Fanuc KAREL source: FanucServiceLib.kl

PROGRAM FANUC_SERVICE_LIB
%NOLOCKGROUP
%NOPAUSE = ERROR + COMMAND + TPENABLE
%NOABORT = ERROR + COMMAND
%COMMENT = 'Shared helpers for resident service'
%ENVIRONMENT sysdef
%ENVIRONMENT kclop
%ENVIRONMENT fdev
%ENVIRONMENT MOTN
%ENVIRONMENT REGOPE
%ENVIRONMENT MULTI
%ENVIRONMENT STRNG

VAR
  g_status  : INTEGER
  g_entry   : INTEGER
  g_bool    : BOOLEAN
  g_int     : INTEGER
  g_real    : REAL
  g_state_real : REAL
  g_state_is_real : BOOLEAN
  g_text1   : STRING[254]
  g_text2   : STRING[254]
  g_text3   : STRING[254]
  g_active_task_name : STRING[36]
  g_target_file : FILE

ROUTINE ClearActiveTask
BEGIN
  g_active_task_name = ''
  SET_INT_REG(98, 1, g_status)
END ClearActiveTask

ROUTINE WriteCallJobTargetFile(target_name : STRING) : BOOLEAN
BEGIN
  SET_FILE_ATR(g_target_file, ATR_IA)
  OPEN FILE g_target_file('rw', 'MD:fanuc_call_job.txt')
  g_status = IO_STATUS(g_target_file)
  IF g_status <> 0 THEN
    RETURN(FALSE)
  ENDIF

  WRITE g_target_file(target_name, CR)
  g_status = IO_STATUS(g_target_file)
  CLOSE FILE g_target_file
  CLR_IO_STAT(g_target_file)

  IF g_status = 0 THEN
    RETURN(TRUE)
  ENDIF
  RETURN(FALSE)
END WriteCallJobTargetFile

ROUTINE WriteOk(ch : FILE; payload : STRING)
BEGIN
  IF payload = '' THEN
    WRITE ch('OK', CR)
  ELSE
    WRITE ch('OK:', payload, CR)
  ENDIF
END WriteOk

ROUTINE WriteErr(ch : FILE; payload : STRING)
BEGIN
  WRITE ch('ERR:', payload, CR)
END WriteErr

ROUTINE WriteCurrentPos(ch : FILE)
VAR
  pos : XYZWPREXT
  raw_pos : XYZWPREXT
  jpos : JOINTPOS
  utool : POSITION
  uframe : POSITION
  out_pos : POSITION
  wjnt_cfg : CONFIG
  ext_ang : ARRAY[3] OF REAL
  reg_status : INTEGER
  kine_status : INTEGER
  config_ref : INTEGER
BEGIN
  DELAY(100)
  raw_pos = CURPOS(0,0)
  jpos = CURJPOS(0,0)
  reg_status = 0
  utool = GET_POS_REG(3, reg_status)
  IF reg_status = 0 THEN
    uframe = GET_POS_REG(4, reg_status)
  ENDIF
  IF reg_status = 0 THEN
    config_ref = 0
    JOINT2POS(jpos, uframe, utool, config_ref, out_pos, wjnt_cfg, ext_ang, kine_status)
    IF kine_status = 0 THEN
      pos = out_pos
    ELSE
      pos = raw_pos
    ENDIF
  ELSE
    pos = raw_pos
  ENDIF
  SET_POS_REG(90, pos, g_status)
  WRITE ch('POS:',
           pos.x::10::3, ',',
           pos.y::10::3, ',',
           pos.z::10::3, ',',
           pos.w::10::3, ',',
           pos.p::10::3, ',',
           pos.r::10::3, CR)
END WriteCurrentPos

ROUTINE WriteCurrentPos00(ch : FILE)
VAR
  pos : XYZWPREXT
  raw_pos : XYZWPREXT
  jpos : JOINTPOS
  utool : POSITION
  uframe : POSITION
  out_pos : POSITION
  wjnt_cfg : CONFIG
  ext_ang : ARRAY[3] OF REAL
  reg_status : INTEGER
  kine_status : INTEGER
  config_ref : INTEGER
BEGIN
  raw_pos = CURPOS(0,0)
  jpos = CURJPOS(0,0)
  reg_status = 0
  utool = GET_POS_REG(3, reg_status)
  IF reg_status = 0 THEN
    uframe = GET_POS_REG(4, reg_status)
  ENDIF
  IF reg_status = 0 THEN
    config_ref = 0
    JOINT2POS(jpos, uframe, utool, config_ref, out_pos, wjnt_cfg, ext_ang, kine_status)
    IF kine_status = 0 THEN
      pos = out_pos
    ELSE
      pos = raw_pos
    ENDIF
  ELSE
    pos = raw_pos
  ENDIF
   SET_POS_REG(91, pos, g_status)
  WRITE ch('POS00:',
           pos.x::10::3, ',',
           pos.y::10::3, ',',
           pos.z::10::3, ',',
           pos.w::10::3, ',',
           pos.p::10::3, ',',
           pos.r::10::3, CR)
END WriteCurrentPos00

ROUTINE WriteCurrentPos001(ch : FILE)
VAR
  pos : XYZWPREXT
BEGIN
  pos = CURPOS(0,0,1)
  WRITE ch('POS001:',
           pos.x::10::3, ',',
           pos.y::10::3, ',',
           pos.z::10::3, ',',
           pos.w::10::3, ',',
           pos.p::10::3, ',',
           pos.r::10::3, CR)
END WriteCurrentPos001

ROUTINE WriteCurrentPos01(ch : FILE)
VAR
  pos : XYZWPREXT
BEGIN
  pos = CURPOS(0,1)
  WRITE ch('POS01:',
           pos.x::10::3, ',',
           pos.y::10::3, ',',
           pos.z::10::3, ',',
           pos.w::10::3, ',',
           pos.p::10::3, ',',
           pos.r::10::3, CR)
END WriteCurrentPos01

ROUTINE WriteCurrentPos10(ch : FILE)
VAR
  pos : XYZWPREXT
BEGIN
  pos = CURPOS(1,0)
  WRITE ch('POS10:',
           pos.x::10::3, ',',
           pos.y::10::3, ',',
           pos.z::10::3, ',',
           pos.w::10::3, ',',
           pos.p::10::3, ',',
           pos.r::10::3, CR)
END WriteCurrentPos10

ROUTINE WriteCurrentPos11(ch : FILE)
VAR
  pos : XYZWPREXT
BEGIN
  pos = CURPOS(1,1)
  WRITE ch('POS11:',
           pos.x::10::3, ',',
           pos.y::10::3, ',',
           pos.z::10::3, ',',
           pos.w::10::3, ',',
           pos.p::10::3, ',',
           pos.r::10::3, CR)
END WriteCurrentPos11

ROUTINE WriteCurrentPos011(ch : FILE)
VAR
  pos : XYZWPREXT
BEGIN
  pos = CURPOS(0,1,1)
  WRITE ch('POS011:',
           pos.x::10::3, ',',
           pos.y::10::3, ',',
           pos.z::10::3, ',',
           pos.w::10::3, ',',
           pos.p::10::3, ',',
           pos.r::10::3, CR)
END WriteCurrentPos011

ROUTINE WriteCurrentPos111(ch : FILE)
VAR
  pos : XYZWPREXT
BEGIN
  pos = CURPOS(1,1,1)
  WRITE ch('POS111:',
           pos.x::10::3, ',',
           pos.y::10::3, ',',
           pos.z::10::3, ',',
           pos.w::10::3, ',',
           pos.p::10::3, ',',
           pos.r::10::3, CR)
END WriteCurrentPos111

ROUTINE WriteCurrentPulse(ch : FILE; axis_count : INTEGER)
VAR
  jpos : JOINTPOS
  vals : ARRAY[9] OF REAL
BEGIN
  vals[1] = 0.0
  vals[2] = 0.0
  vals[3] = 0.0
  vals[4] = 0.0
  vals[5] = 0.0
  vals[6] = 0.0

  jpos = CURJPOS(0,0)
  CNV_JPOS_REL(jpos, vals, g_status)
  IF g_status <> 0 THEN
    WriteErr(ch, 'GET_PULSE_FAIL')
    RETURN
  ENDIF

  IF axis_count <= 6 THEN
    WRITE ch('PULSE:',
             vals[1]::10::3, ',',
             vals[2]::10::3, ',',
             vals[3]::10::3, ',',
             vals[4]::10::3, ',',
             vals[5]::10::3, ',',
             vals[6]::10::3, ',',
             0.0::10::3, ',',
             0.0::10::3, ',',
             0.0::10::3, CR)
    RETURN
  ENDIF

  IF axis_count = 7 THEN
    WRITE ch('PULSE:',
             vals[1]::10::3, ',',
             vals[2]::10::3, ',',
             vals[3]::10::3, ',',
             vals[4]::10::3, ',',
             vals[5]::10::3, ',',
             vals[6]::10::3, ',',
             vals[7]::10::3, ',',
             0.0::10::3, ',',
             0.0::10::3, CR)
    RETURN
  ENDIF

  IF axis_count = 8 THEN
    WRITE ch('PULSE:',
             vals[1]::10::3, ',',
             vals[2]::10::3, ',',
             vals[3]::10::3, ',',
             vals[4]::10::3, ',',
             vals[5]::10::3, ',',
             vals[6]::10::3, ',',
             vals[7]::10::3, ',',
             vals[8]::10::3, ',',
             0.0::10::3, CR)
    RETURN
  ENDIF

  WRITE ch('PULSE:',
           vals[1]::10::3, ',',
           vals[2]::10::3, ',',
           vals[3]::10::3, ',',
           vals[4]::10::3, ',',
           vals[5]::10::3, ',',
           vals[6]::10::3, ',',
           vals[7]::10::3, ',',
           vals[8]::10::3, ',',
           vals[9]::10::3, CR)
END WriteCurrentPulse

ROUTINE WriteDoneState(ch : FILE)
VAR
  moving : BOOLEAN
  task_name : STRING[36]
  task_no : INTEGER
  task_status : INTEGER
  task_dummy : STRING[2]
  task_query_status : INTEGER
BEGIN
  GET_VAR(g_entry, '*SYSTEM*', '$MOR_GRP[1].$ROB_MOVE', moving, g_status)
  IF g_status = 0 THEN
    IF moving THEN
      WRITE ch('DONE:0', CR)
    ELSE
      IF g_active_task_name = '' THEN
        WRITE ch('DONE:1', CR)
        RETURN
      ENDIF

      -- ROB_MOVE=FALSE 只表示采样瞬间没有轴运动；任务仍可能处于等待、暂停、
      -- 接受或减速中。只有任务查询明确到达 PG_ABORTED 才能释放高层租约。
      task_name = g_active_task_name
      task_no = 0
      GET_TSK_INFO(task_name, task_no, TSK_STATUS,
                   task_status, task_dummy, task_query_status)
      IF task_query_status <> 0 THEN
        WRITE ch('DONE:-1', CR)
        RETURN
      ENDIF
      IF task_status = PG_ABORTED THEN
        ClearActiveTask
        WRITE ch('DONE:1', CR)
      ELSE
        WRITE ch('DONE:0', CR)
      ENDIF
    ENDIF
  ELSE
    WRITE ch('DONE:-1', CR)
  ENDIF
END WriteDoneState

ROUTINE FindChar(src : STRING; token : STRING) : INTEGER
VAR
  i   : INTEGER
  one : STRING[1]
BEGIN
  FOR i = 1 TO STR_LEN(src) DO
    one = SUB_STR(src, i, 1)
    IF one = token THEN
      RETURN(i)
    ENDIF
  ENDFOR
  RETURN(0)
END FindChar

ROUTINE Payload(cmd : STRING; prefix_len : INTEGER; out_str : STRING)
BEGIN
  out_str = SUB_STR(cmd, prefix_len + 1, STR_LEN(cmd) - prefix_len)
END Payload

ROUTINE DoSetInt(ch : FILE; cmd : STRING)
VAR
  comma_pos : INTEGER
  reg_name  : STRING[64]
  reg_value : STRING[64]
  reg_index : INTEGER
BEGIN
  Payload(cmd, 8, g_text1)
  comma_pos = FindChar(g_text1, ',')
  IF comma_pos <= 1 THEN
    WriteErr(ch, 'BAD_SET_INT')
    RETURN
  ENDIF

  reg_name = SUB_STR(g_text1, 1, comma_pos - 1)
  reg_value = SUB_STR(g_text1, comma_pos + 1, STR_LEN(g_text1) - comma_pos)

  IF SUB_STR(reg_name, 1, 3) = 'INT' THEN
    CNV_STR_INT(SUB_STR(reg_name, 4, STR_LEN(reg_name) - 3), reg_index)
  ELSE
    IF reg_name = 'WELD_TRACK_NO' THEN
      reg_index = 30
    ELSE
      WriteErr(ch, 'UNSUPPORTED_INT_NAME')
      RETURN
    ENDIF
  ENDIF

  CNV_STR_INT(reg_value, g_int)
  SET_INT_REG(reg_index, g_int, g_status)
  IF g_status = 0 THEN
    WriteOk(ch, '')
  ELSE
    WriteErr(ch, 'SET_INT_FAIL')
  ENDIF
END DoSetInt

ROUTINE DoGetInt(ch : FILE; cmd : STRING)
VAR
  comma_pos : INTEGER
  reg_type  : STRING[16]
  reg_index : INTEGER
BEGIN
  Payload(cmd, 8, g_text1)
  comma_pos = FindChar(g_text1, ',')
  IF comma_pos <= 0 THEN
    WriteErr(ch, 'BAD_GET_INT')
    RETURN
  ENDIF

  reg_type = SUB_STR(g_text1, 1, comma_pos - 1)
  IF reg_type <> 'INT' THEN
    WriteErr(ch, 'UNSUPPORTED_GET_INT')
    RETURN
  ENDIF

  CNV_STR_INT(SUB_STR(g_text1, comma_pos + 1, STR_LEN(g_text1) - comma_pos), reg_index)
  GET_REG(reg_index, g_bool, g_int, g_real, g_status)
  IF g_status = 0 THEN
    IF g_bool THEN
      WRITE ch('INT:', g_real::10::3, CR)
    ELSE
      WRITE ch('INT:', g_int, CR)
    ENDIF
  ELSE
    WriteErr(ch, 'GET_INT_FAIL')
  ENDIF
END DoGetInt

ROUTINE DoCallJob(ch : FILE; cmd : STRING)
BEGIN
  Payload(cmd, 9, g_text1)
  -- 先把被动完成寄存器置为运行态，再接受任务；这样 S5 不会在 RUN_TASK
  -- 已接受但 g_active_task_name 尚未写入的窗口误报完成。
  SET_INT_REG(98, 0, g_status)
  IF g_status <> 0 THEN
    WriteErr(ch, 'CALL_JOB_STATE_FAIL')
    RETURN
  ENDIF
  RUN_TASK(g_text1, 1, FALSE, FALSE, 1, g_status)
  IF g_status = 0 THEN
    g_active_task_name = g_text1
    WriteOk(ch, '')
  ELSE
    ClearActiveTask
    WriteErr(ch, 'CALL_JOB_FAIL')
  ENDIF
END DoCallJob

ROUTINE DoProgramStop(ch : FILE)
VAR
  task_name : STRING[36]
  abort_status : INTEGER
  task_no : INTEGER
  task_status : INTEGER
  task_dummy : STRING[2]
  task_query_status : INTEGER
BEGIN
  task_name = g_active_task_name
  IF task_name = '' THEN
    WriteErr(ch, 'NO_ACTIVE_CALL_JOB')
    RETURN
  ENDIF

  -- 任务可能刚好在用户按 STOP 前自然结束。先确认终态，避免对已经
  -- PG_ABORTED 的任务再次 ABORT_TASK 返回错误并留下无法解除的闭锁。
  task_no = 0
  GET_TSK_INFO(task_name, task_no, TSK_STATUS,
               task_status, task_dummy, task_query_status)
  IF (task_query_status = 0) AND (task_status = PG_ABORTED) THEN
    ClearActiveTask
    WriteOk(ch, 'ALREADY_STOPPED')
    RETURN
  ENDIF

  -- force_sw=TRUE：即使目标任务设置 ignore-abort 也中止；
  -- cancel_mtn_sw=TRUE：同步取消该任务所属运动组的当前/排队运动。
  ABORT_TASK(task_name, TRUE, TRUE, abort_status)
  IF abort_status = 0 THEN
    -- ABORT_TASK 成功只代表中止请求被接受；ABORTING/减速期间继续保持
    -- active name 和 R[98]=0，由 WriteDoneState 的 PG_ABORTED 回读最终清除。
    WriteOk(ch, 'ABORT_REQUESTED')
  ELSE
    WriteErr(ch, 'PROGRAM_STOP_FAIL')
  ENDIF
END DoProgramStop

ROUTINE DoSetTpSpeed(ch : FILE; cmd : STRING)
BEGIN
  Payload(cmd, 13, g_text1)
  CNV_STR_INT(g_text1, g_int)
  SET_INT_REG(17, g_int, g_status)
  IF g_status = 0 THEN
    WriteOk(ch, '')
  ELSE
    WriteErr(ch, 'SET_TP_SPEED_FAIL')
  ENDIF
END DoSetTpSpeed

ROUTINE DoStopService(ch : FILE)
BEGIN
  SET_INT_REG(99, 1, g_status)
  IF g_status = 0 THEN
    WriteOk(ch, 'STOPPING')
  ELSE
    WriteErr(ch, 'STOP_SERVICE_FAIL')
  ENDIF
END DoStopService

ROUTINE PopToken(rest : STRING; token : STRING)
VAR
  comma_pos : INTEGER
BEGIN
  comma_pos = FindChar(rest, ',')
  IF comma_pos <= 0 THEN
    token = rest
    rest = ''
  ELSE
    token = SUB_STR(rest, 1, comma_pos - 1)
    rest = SUB_STR(rest, comma_pos + 1, STR_LEN(rest) - comma_pos)
  ENDIF
END PopToken

ROUTINE DoSetPosVar(ch : FILE; cmd : STRING)
VAR
  cmd_body : STRING[254]
  token    : STRING[64]
  reg_no   : INTEGER
  pos_type : INTEGER
  idx      : INTEGER
  vals     : ARRAY[9] OF REAL
  xyz_pos  : XYZWPR
  jnt_pos  : JOINTPOS
  xyz_cfg  : CONFIG
BEGIN
  Payload(cmd, 12, cmd_body)

  PopToken(cmd_body, token)
  CNV_STR_INT(token, reg_no)
  PopToken(cmd_body, token)
  CNV_STR_INT(token, pos_type)

  FOR idx = 1 TO 9 DO
    vals[idx] = 0.0
  ENDFOR

  FOR idx = 1 TO 8 DO
    PopToken(cmd_body, token)
    CNV_STR_REAL(token, vals[idx])
  ENDFOR

  IF pos_type = 0 THEN
    xyz_pos = CURPOS(0, 0)
    xyz_pos.x = vals[1]
    xyz_pos.y = vals[2]
    xyz_pos.z = vals[3]
    xyz_pos.w = vals[4]
    xyz_pos.p = vals[5]
    xyz_pos.r = vals[6]
    CNV_STR_CONF('N U T, 0, 0, 0', xyz_cfg, g_status)
    IF g_status <> 0 THEN
      WriteErr(ch, 'BAD_CONFIG')
      RETURN
    ENDIF
    xyz_pos.config_data = xyz_cfg
    SET_POS_REG(reg_no, xyz_pos, g_status)
  ELSE
    CNV_REL_JPOS(vals, jnt_pos, g_status)
    IF g_status <> 0 THEN
      WriteErr(ch, 'BAD_JPOS')
      RETURN
    ENDIF
    SET_JPOS_REG(reg_no, jnt_pos, g_status)
  ENDIF

  IF g_status = 0 THEN
    WriteOk(ch, '')
  ELSE
    WriteErr(ch, 'SET_POS_VAR_FAIL')
  ENDIF
END DoSetPosVar

ROUTINE DoGetPosVar(ch : FILE; cmd : STRING)
VAR
  cmd_body : STRING[254]
  token    : STRING[64]
  reg_no   : INTEGER
  move_type : INTEGER
  pos_type : INTEGER
  num_axes : INTEGER
  pos      : XYZWPREXT
  cfg_text : STRING[32]
BEGIN
  Payload(cmd, 12, cmd_body)

  PopToken(cmd_body, token)
  CNV_STR_INT(token, reg_no)
  PopToken(cmd_body, token)
  CNV_STR_INT(token, move_type)

  POS_REG_TYPE(reg_no, 1, pos_type, num_axes, g_status)
  IF g_status <> 0 THEN
    WriteErr(ch, 'GET_POS_TYPE_FAIL')
    RETURN
  ENDIF

  pos = GET_POS_REG(reg_no, g_status, 1)
  IF g_status <> 0 THEN
    WriteErr(ch, 'GET_POS_REG_FAIL')
    RETURN
  ENDIF

  CNV_CONF_STR(pos.config_data, cfg_text)
  WRITE ch('POSVAR:',
           reg_no, ',',
           pos_type, ',',
           num_axes, ',',
           pos.x::10::3, ',',
           pos.y::10::3, ',',
           pos.z::10::3, ',',
           pos.w::10::3, ',',
           pos.p::10::3, ',',
           pos.r::10::3, ',',
           cfg_text, CR)
END DoGetPosVar

ROUTINE DispatchCommand(ch : FILE; cmd : STRING)
BEGIN
  IF cmd = 'HELLO' THEN
    WriteOk(ch, 'READY')
    RETURN
  ENDIF

  IF cmd = 'CHECK_DONE' THEN
    WriteDoneState(ch)
    RETURN
  ENDIF
  IF cmd = 'GET_CUR_POS' THEN
    WriteCurrentPos(ch)
    RETURN
  ENDIF
  IF cmd = 'GET_CUR_POS_00' THEN
    WriteCurrentPos00(ch)
    RETURN
  ENDIF
  IF cmd = 'GET_CUR_POS_001' THEN
    WriteCurrentPos001(ch)
    RETURN
  ENDIF
  IF cmd = 'GET_CUR_POS_01' THEN
    WriteCurrentPos01(ch)
    RETURN
  ENDIF
  IF cmd = 'GET_CUR_POS_10' THEN
    WriteCurrentPos10(ch)
    RETURN
  ENDIF
  IF cmd = 'GET_CUR_POS_11' THEN
    WriteCurrentPos11(ch)
    RETURN
  ENDIF
  IF cmd = 'GET_CUR_POS_011' THEN
    WriteCurrentPos011(ch)
    RETURN
  ENDIF
  IF cmd = 'GET_CUR_POS_111' THEN
    WriteCurrentPos111(ch)
    RETURN
  ENDIF
  IF cmd = 'GET_CUR_PULSE' THEN
    WriteCurrentPulse(ch, 6)
    RETURN
  ENDIF
  IF SUB_STR(cmd, 1, 14) = 'GET_CUR_PULSE:' THEN
    Payload(cmd, 14, g_text1)
    CNV_STR_INT(g_text1, g_int)
    WriteCurrentPulse(ch, g_int)
    RETURN
  ENDIF
  IF cmd = 'GET_USER_PROGRAM' THEN
    WRITE ch('PROGRAM:FANUC_RESIDENT_SERVICE;LIB=20260710_ABORT_TASK_STATE_V2', CR)
    RETURN
  ENDIF
  IF cmd = 'GET_USER_PROJECT' THEN
    WRITE ch('PROJECT:MD', CR)
    RETURN
  ENDIF
  IF SUB_STR(cmd, 1, 8) = 'SET_INT:' THEN
    DoSetInt(ch, cmd)
    RETURN
  ENDIF
  IF SUB_STR(cmd, 1, 8) = 'GET_INT:' THEN
    DoGetInt(ch, cmd)
    RETURN
  ENDIF
  IF SUB_STR(cmd, 1, 9) = 'CALL_JOB:' THEN
    DoCallJob(ch, cmd)
    RETURN
  ENDIF
  IF SUB_STR(cmd, 1, 13) = 'SET_TP_SPEED:' THEN
    DoSetTpSpeed(ch, cmd)
    RETURN
  ENDIF
  IF cmd = 'STOP_SERVICE' THEN
    DoStopService(ch)
    RETURN
  ENDIF
  IF SUB_STR(cmd,1,9) = 'SET_REAL:' THEN
    WriteOk(ch, '')
    RETURN
  ENDIF
  IF SUB_STR(cmd,1,12) = 'SET_POS_VAR:' THEN
    DoSetPosVar(ch, cmd)
    RETURN
  ENDIF
  IF SUB_STR(cmd,1,12) = 'GET_POS_VAR:' THEN
    DoGetPosVar(ch, cmd)
    RETURN
  ENDIF
  IF SUB_STR(cmd,1,10) = 'SET_SPEED:' THEN
    WriteOk(ch, '')
    RETURN
  ENDIF
  IF SUB_STR(cmd,1,18) = 'LOAD_USER_PROGRAM:' THEN
    WriteOk(ch, '')
    RETURN
  ENDIF
  IF cmd = 'UNLOAD_USER_PROGRAM' THEN
    WriteOk(ch, '')
    RETURN
  ENDIF
  IF cmd = 'PROGRAM_START' THEN
    WriteOk(ch, '')
    RETURN
  ENDIF
  IF cmd = 'PROGRAM_STOP' THEN
    DoProgramStop(ch)
    RETURN
  ENDIF
  IF cmd = 'SERVO_ON' THEN
    WriteOk(ch, '')
    RETURN
  ENDIF
  IF cmd = 'SERVO_OFF' THEN
    WriteOk(ch, '')
    RETURN
  ENDIF
  IF cmd = 'CLEAR_ALARM' THEN
    WriteOk(ch, '')
    RETURN
  ENDIF
  IF SUB_STR(cmd,1,13) = 'SET_SYS_MODE:' THEN
    WriteOk(ch, '')
    RETURN
  ENDIF
  IF SUB_STR(cmd,1,12) = 'SET_TOOL_NO:' THEN
    WriteOk(ch, '')
    RETURN
  ENDIF
  IF SUB_STR(cmd,1,14) = 'GET_TOOL_DATA:' THEN
    WriteOk(ch, '')
    RETURN
  ENDIF
  IF SUB_STR(cmd,1,16) = 'AXIS_PULSE_MOVE:' THEN
    WriteOk(ch, '')
    RETURN
  ENDIF
  IF SUB_STR(cmd,1,9) = 'POS_MOVE:' THEN
    WriteOk(ch, '')
    RETURN
  ENDIF
  IF SUB_STR(cmd,1,17) = 'MOVE_BY_JOB_AXIS:' THEN
    WriteOk(ch, '')
    RETURN
  ENDIF
  IF SUB_STR(cmd,1,16) = 'MOVE_BY_JOB_POS:' THEN
    WriteOk(ch, '')
    RETURN
  ENDIF
  IF SUB_STR(cmd,1,19) = 'MOVE_BY_JOB_VECTOR:' THEN
    WriteOk(ch, '')
    RETURN
  ENDIF

  WriteErr(ch, 'UNKNOWN_CMD')
END DispatchCommand

BEGIN
END FANUC_SERVICE_LIB
